// TwinCAT 3 PLC project PizzaProject
// ProgramVersion: 3.1.4023.0
// libraries:
//   VisuElemMeter, 3.5.4.0 (System)
//   VisuElems, 3.5.4.10 (System)
//   VisuElemsSpecialControls, 3.5.4.10 (System)
//   VisuElemsWinControls, 3.5.4.10 (System)
//   VisuElemTextEditor, 3.5.4.0 (System)
//   visuinputs, 3.5.4.0 (system)
//   VisuNativeControl, 3.5.4.0 (System)
//   Tc2_Standard, * (Beckhoff Automation GmbH)
//   Tc2_System, * (Beckhoff Automation GmbH)
//   Tc2_Utilities, * (Beckhoff Automation GmbH)
//   Tc3_Module, * (Beckhoff Automation GmbH)
//   VisuDialogs, * (System)
// project tree:
//   DUTs/ E_PIZZA_TYPES.TcDUT (not stored), ST_PIZZA.TcDUT
//   / GlobalTextList.TcGTLO, PlcTask.TcTTO (not stored), Visualization Manager.TcVMO (not stored)
//   GVLs/ HMI_VARS.TcGVL
//   POUs/ MAIN.TcPOU, FB_PIZZA_OVEN.TcPOU, F_FIFO_WRITE.TcPOU
//   VISUs/ Visualization.TcVIS

// ---- DUTs/ST_PIZZA.TcDUT
TYPE ST_PIZZA :
STRUCT
	bExist : BOOL;
	dtTimeEnteredOven : DATE_AND_TIME;
	dtTimeExitedOven : DATE_AND_TIME;
	tTimeInOven : TIME;
	eType : E_PIZZA_TYPES; // 0 = Cheese, 1 = Pep, 2 = sausage
	
END_STRUCT
END_TYPE

// ---- GVLs/HMI_VARS.TcGVL
VAR_GLOBAL

	iState : DINT; // My machine state.
	bStartButton : BOOL;
	
	arrPizzaHistory : ARRAY [0..100] OF ST_PIZZA;
	
	fbNT_GetTime : GETSYSTEMTIME;
	stCurrentTime : T_FILETIME;
	dtCurrentTime : DATE_AND_TIME;
END_VAR

// ---- POUs/MAIN.TcPOU
PROGRAM MAIN
VAR

	fbMyPizzaOven : FB_PIZZA_OVEN;  // My Instance of oven 1
	
	bLoadPizza : BOOL;  // put a pizza on the input side
	bRemovePizza : BOOL;  // take pizza off output side.
	stFileTime : T_FILETIME;
	
	i : DINT;  
	
	arrMyBools : ARRAY [0..100] OF STRING;
	
	fbMyTimer : TON; 
	
END_VAR

VAR CONSTANT
	MAX_OVENS : DINT := 1; // This is 2.. 
END_VAR


fbMyPizzaOven(bLoadPizza:=bLoadPizza , bRemovePizza:=bRemovePizza );

fbMyTimer(IN:=NOT fbMyTimer.Q, PT:=T#100MS);

fbNT_GetTime(timeLoDW => stFileTime.dwLowDateTime,
			timeHiDW => stFileTime.dwHighDateTime);
			
dtCurrentTime := FILETIME_TO_DT(fileTime := stFileTime);

END_PROGRAM

// ---- POUs/FB_PIZZA_OVEN.TcPOU
FUNCTION_BLOCK FB_PIZZA_OVEN
VAR_INPUT
	bLoadPizza : BOOL;  // put a pizza on the input side
	bRemovePizza : BOOL;  // take pizza off output side.
END_VAR
VAR_OUTPUT
	iTotalPizzasCooked : UDINT;			
	bBuzzer : BOOL;
	bLight : BOOL;  // NEW!
END_VAR
VAR

	fbLoad_RTRIG : R_TRIG;
	fbRemove_RTRIG : R_TRIG;

	iState : DINT;
	iLastState : DINT;
	sStateDesc : STRING;

	//timers
	fbMyTimer : TON;  // My Timer... for stuff.
	
	stPizzaOnDeck : ST_PIZZA; // Location of possible pizza... 
	stPizzaInOven : ST_PIZZA;  
	stPizzaDone   : ST_PIZZA; 
	
	arrStateDescHistory : ARRAY [1..100] OF STRING;

END_VAR
VAR CONSTANT
	stNULL_PIZZA : ST_PIZZA;  
END_VAR

// If there is room
IF stPizzaOnDeck.bExist AND NOT stPizzaInOven.bExist THEN
	stPizzaInOven := stPizzaOnDeck;
	stPizzaOnDeck := stNULL_PIZZA;  // Remove pizza.
END_IF


// Handle buttons... / sim inputs
fbLoad_RTRIG(clk := bLoadPizza);
IF fbLoad_RTRIG.Q THEN
	//bLoadPizza := FALSE;
	stPizzaOnDeck.bExist := TRUE;
	stPizzaOnDeck.eType := eType_Sausage;
END_IF

fbRemove_RTRIG(clk := bRemovePizza);
IF fbRemove_RTRIG.Q THEN
	F_FIFO_WRITE(cbData := SIZEOF(stPizzaDone), pData := ADR(stPizzaDone),
					cbBuffer := SIZEOF(arrPizzaHistory), pBuffer := ADR(arrPizzaHistory)
	);
	stPizzaDone := stNULL_PIZZA;
	//bRemovePizza := FALSE;
END_IF

CASE iState OF
	
	0:  // Wait for pizza in oven.
		sStateDesc := 'Waiting on Pizza Now.';
		IF stPizzaInOven.bExist THEN
			stPizzaInOven.dtTimeEnteredOven := dtCurrentTime;
			iState := 10;
		END_IF

	10: // We just got a pizza! Cook it.
		sStateDesc := 'Baking That Pizza Now.';
		fbMyTimer(IN:=TRUE,PT:=T#3S);
		IF fbMyTimer.Q THEN
			fbMyTimer(IN:=FALSE);
			iState := 20;	
		END_IF
 	
	
	20: // Can we move the pizza out of the oven?  Its going to burn.
	
		sStateDesc := 'PIZZA BURNING!!!!.';
	
		IF NOT stPizzaDone.bExist THEN
		
			//Simulate conveyor.
			stPizzaInOven.dtTimeExitedOven := dtCurrentTime;
			stPizzaDone := stPizzaInOven;
			stPizzaInOven := stNULL_PIZZA;
			bBuzzer := FALSE;
	
			iState := 30;
	
		ELSE
			
			bBuzzer := TRUE;
			
		END_IF
	
	30:  // Pizza just removed. on output tray.
	
		stPizzaDone.tTimeInOven := stPizzaDone.dtTimeExitedOven - stPizzaDone.dtTimeEnteredOven; 
		iTotalPizzasCooked := iTotalPizzasCooked + 1;
		iState := 0;   // Go wait for new pizza in oven!!

	
ELSE
	
	sStateDesc := 'Invalid state!';

END_CASE


// Start state history:

IF iLastState <> iState THEN

	// Do stuff here to log transitions.... 
	F_FIFO_WRITE(cbData := SIZEOF(sStateDesc), pData := ADR(sStateDesc),
					cbBuffer := SIZEOF(arrStateDescHistory), pBuffer := ADR(arrStateDescHistory)
	);
	
	// Reset for next time.
	iLastState := iState;

END_IF

END_FUNCTION_BLOCK

// ---- POUs/F_FIFO_WRITE.TcPOU
FUNCTION F_FIFO_WRITE : BOOL
VAR_INPUT
	cbData : UDINT;
	pData : POINTER TO BYTE;
	
	cbBuffer : UDINT;
	pBuffer : POINTER TO BYTE;
END_VAR
VAR
END_VAR



FW_MemMove(pDest := pBuffer + cbData, pSrc := pBuffer, cbLen := cbBuffer - cbData);


FW_MemMove(pDest := pBuffer, pSrc := pData, cbLen := cbData);

END_FUNCTION

// ---- GlobalTextList.TcGTLO
TEXTLIST GlobalTextList
  13 = 'B'
  7 = 'Buzzer'
  271 = 'Czy pizza została wykonana?'
  933 = 'Czy pizza została wypieczona?'
  525 = 'Data i godzina rozpoczęcia pieczenia pizzy'
  728 = 'Data i godzina zakończenia pieczenia pizzy'
  226 = 'Data rozpoczęcia pieczenia pizzy'
  746 = 'Długość pieczenia pizzy'
  2 = 'Elapsed Tiime: %s'
  5 = 'Elapsed Time: '
  6 = 'Elapsed Time: %s'
  1 = 'Insert Pizza'
  3 = 'Insert Pizza '
  14 = 'L'
  8 = 'Light'
  12 = 'New Pizza Ready'
  528 = 'Nowa pizza'
  11 = 'Package Pizza'
  0 = 'Pizza'
  10 = 'Pizza (Done)'
  364 = 'Pizza (na stole)'
  9 = 'Pizza (On Deck)'
  343 = 'Pizza (w piecu)'
  490 = 'Pizza (wykonana)'
  16 = 'Pizzas Cooked %d'
  15 = 'Pizzas Cooked %I'
  17 = 'Pizzas Cooked: %d'
  424 = 'Spakuj pizze'
  18 = 'Status: %s'
  4 = 'Take Pizza Out'
  466 = 'Typ pizzy'
  450 = 'Upieczone pizze: %d'
  910 = 'Upłynięty czas: %s'
  37 = 'Zapakuj pizze'
END_TEXTLIST

// ---- VISUs/Visualization.TcVIS
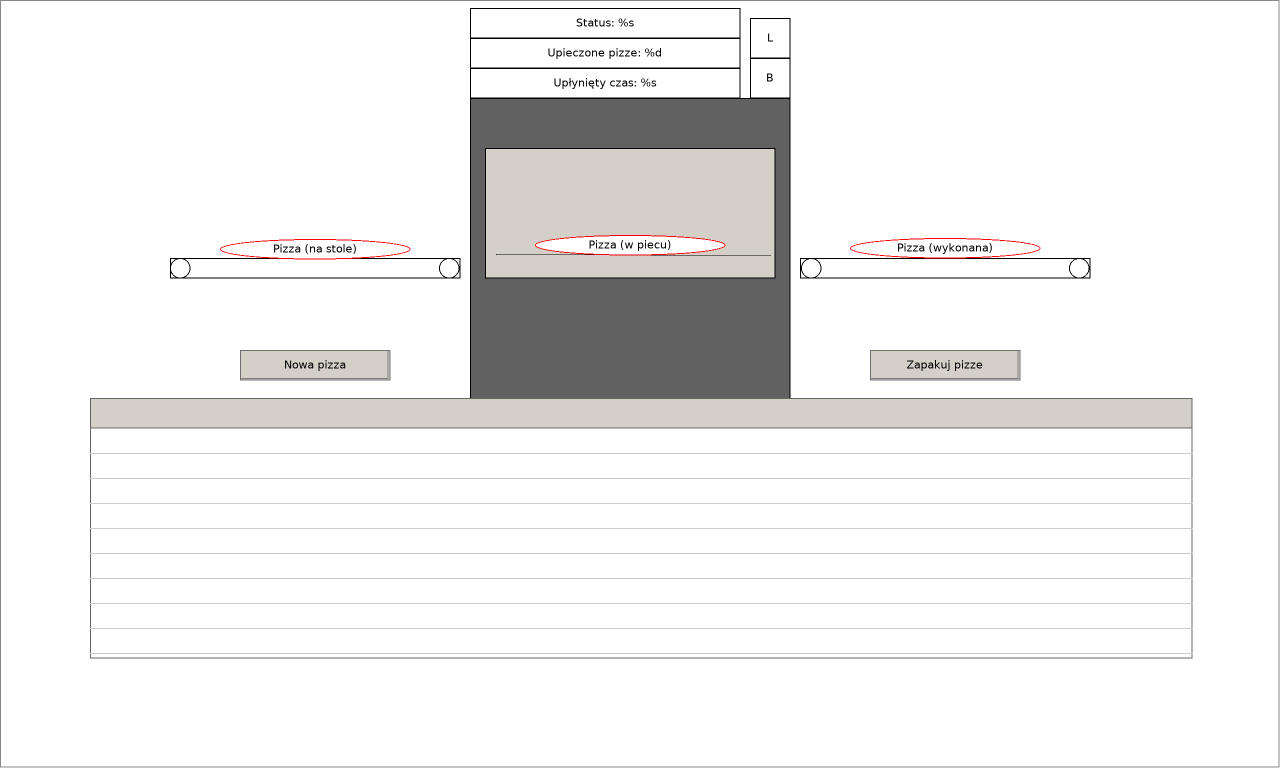
VISUALIZATION Visualization  // 1280x768
    Rectangle (470,98 320x480)
    Button (240,350 150x30), "Nowa pizza"
        tap MAIN.bLoadPizza
    Button (870,350 150x30), "Zapakuj pizze"
        tap MAIN.bRemovePizza
    Button (663,152 18x0)
    Rectangle (485,148 290x130)
    Rectangle (470,68 270x30), "Upłynięty czas: %s", text variable: MAIN.fbMyPizzaOven.fbMyTimer.ET
    RoundedRectangle (170,258 290x20)
    RoundedRectangle (800,258 290x20)
    Ellipse (850,238 190x20), "Pizza (wykonana)", invisible if: NOT MAIN.fbMyPizzaOven.stPizzaDone.bExist
    Ellipse (220,239 190x20), "Pizza (na stole)", invisible if: NOT MAIN.fbMyPizzaOven.stPizzaOnDeck.bExist
    Line (496,254) (770,255)
    Ellipse (535,235 190x20), "Pizza (w piecu)", invisible if: NOT MAIN.fbMyPizzaOven.stPizzaInOven.bExist
    RoundedRectangle (750,58 40x40), "B", colour toggle: MAIN.fbMyPizzaOven.bBuzzer
    RoundedRectangle (750,18 40x40), "L", colour toggle: MAIN.fbMyPizzaOven.bLight
    Rectangle (470,38 270x30), "Upieczone pizze: %d", text variable: MAIN.fbMyPizzaOven.iTotalPizzasCooked
    Ellipse (170,258 20x20)
    Ellipse (439,258 20x20)
    Rectangle (470,8 270x30), "Status: %s", text variable: MAIN.fbMyPizzaOven.sStateDesc
    Table (90,398 1102x260), data array: HMI_VARS.arrPizzaHistory
        p3854506369: HMI_VARS.arrPizzaHistory[INDEX].bExist
        p1892666644: HMI_VARS.arrPizzaHistory[INDEX].dtTimeEnteredOven
        p338671338: HMI_VARS.arrPizzaHistory[INDEX].dtTimeExitedOven
        p2170511999: HMI_VARS.arrPizzaHistory[INDEX].tTimeInOven
        p3723444502: HMI_VARS.arrPizzaHistory[INDEX].eType
        p2232123230: Czy pizza została wypieczona?
        p511219082: Data i godzina rozpoczęcia pieczenia pizzy
        p1755163831: Data i godzina zakończenia pieczenia pizzy
        p4092479075: Długość pieczenia pizzy
        p2237128397: Typ pizzy
    Ellipse (801,258 20x20)
    Ellipse (1069,258 20x20)
END_VISUALIZATION
